// TIA Portal V19 export
TYPE "PPrf_Pivot"
// stored: Access Published
   STRUCT
      PrgNo : DInt;
      PrgName : String[79];
      RecordNo : Int;   // Record Number: 1..PPRF_TOTAL_ARCHIVE_ITEMS
   END_STRUCT;
END_TYPE
